TYPE csp_transfer_infeed_accumulation_level_enum :(
	CSP_TRANSFER_INFEED_ACCUMULATION_LEVEL_STATUS_IDLE						:= 0,
	CSP_TRANSFER_INFEED_ACCUMULATION_LEVEL_STATUS_EMPTYING					:= 1,
	CSP_TRANSFER_INFEED_ACCUMULATION_LEVEL_STATUS_EMPTYING_UNDER_MIN_DELAY	:= 2,
	CSP_TRANSFER_INFEED_ACCUMULATION_LEVEL_STATUS_EMPTY						:= 3,
	CSP_TRANSFER_INFEED_ACCUMULATION_LEVEL_STATUS_UNDER_MIN					:= 4,
	CSP_TRANSFER_INFEED_ACCUMULATION_LEVEL_STATUS_MIN						:= 5,
	CSP_TRANSFER_INFEED_ACCUMULATION_LEVEL_STATUS_LOW						:= 6,
	CSP_TRANSFER_INFEED_ACCUMULATION_LEVEL_STATUS_NORMAL					:= 7,
	CSP_TRANSFER_INFEED_ACCUMULATION_LEVEL_STATUS_JAM						:= 8,
	CSP_TRANSFER_INFEED_ACCUMULATION_LEVEL_STATUS_INCOHERENT				:= 9,
	CSP_TRANSFER_INFEED_ACCUMULATION_LEVEL_STATUS_ERROR						:= 100
    ) := CSP_TRANSFER_INFEED_ACCUMULATION_LEVEL_STATUS_IDLE;
END_TYPE

(* stored: Version 1.1.0.1, ProductVersion 3.1.4024.3
   DUT csp_transfer_infeed_accumulation_level_enum: Id {7c9d60a7-31b3-4761-ade4-887908322511} *)
